FUNCTION_BLOCK InputPipe (* Composite Function Block Type *)
  (* Standard: 61499-2 *)
  (* Version 0.0, 2011-12-23, 4DIAC-IDE, 4DIAC-Consortium *)
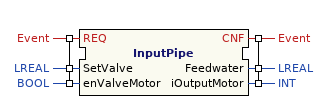
  EVENT_INPUT
    REQ WITH SetValve, enValveMotor; (* Normal Execution Request *)
  END_EVENT
  EVENT_OUTPUT
    CNF WITH Feedwater, iOutputMotor; (* Execution Confirmation *)
  END_EVENT
  VAR_INPUT
    SetValve : LREAL; (* Input event qualifier *)
    enValveMotor : BOOL;
  END_VAR
  VAR_OUTPUT
    Feedwater : LREAL; (* Output event qualifier *)
    iOutputMotor : INT;
  END_VAR
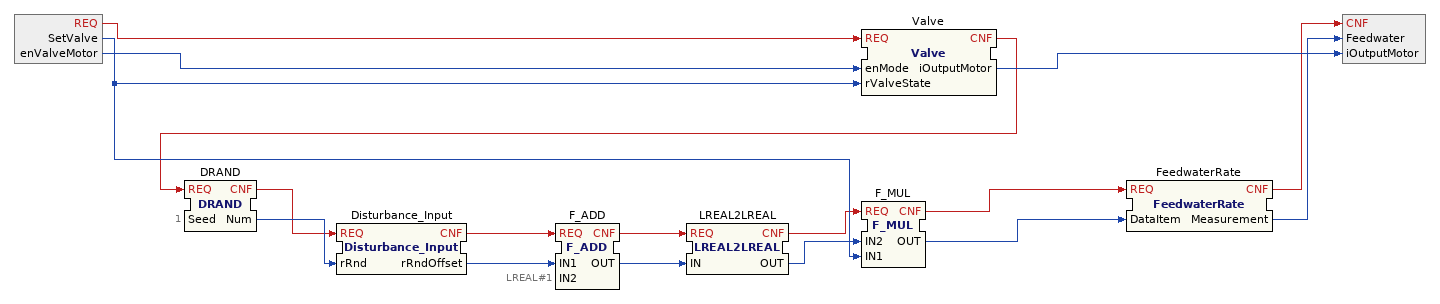
  FBS
    DRAND : DRAND(Seed := 1);
    Valve : Valve;
    FeedwaterRate : FeedwaterRate;
    Disturbance_Input : Disturbance_Input;
    F_MUL : F_MUL;
    F_ADD : F_ADD(IN2 := LREAL#1);
    LREAL2LREAL : LREAL2LREAL;
  END_FBS
  EVENT_CONNECTIONS
    REQ TO Valve.REQ;
    Valve.CNF TO DRAND.REQ;
    FeedwaterRate.CNF TO CNF;
    DRAND.CNF TO Disturbance_Input.REQ;
    Disturbance_Input.CNF TO F_ADD.REQ;
    F_ADD.CNF TO LREAL2LREAL.REQ;
    LREAL2LREAL.CNF TO F_MUL.REQ;
    F_MUL.CNF TO FeedwaterRate.REQ;
  END_CONNECTIONS
  DATA_CONNECTIONS
    SetValve TO Valve.rValveState;
    enValveMotor TO Valve.enMode;
    FeedwaterRate.Measurement TO Feedwater;
    Valve.iOutputMotor TO iOutputMotor;
    DRAND.Num TO Disturbance_Input.rRnd;
    Disturbance_Input.rRndOffset TO F_ADD.IN1;
    F_ADD.OUT TO LREAL2LREAL.IN;
    LREAL2LREAL.OUT TO F_MUL.IN2;
    F_MUL.OUT TO FeedwaterRate.DataItem;
    SetValve TO F_MUL.IN1;
  END_CONNECTIONS
END_FUNCTION_BLOCK
